ABB RAPID module: PathProbe.mod

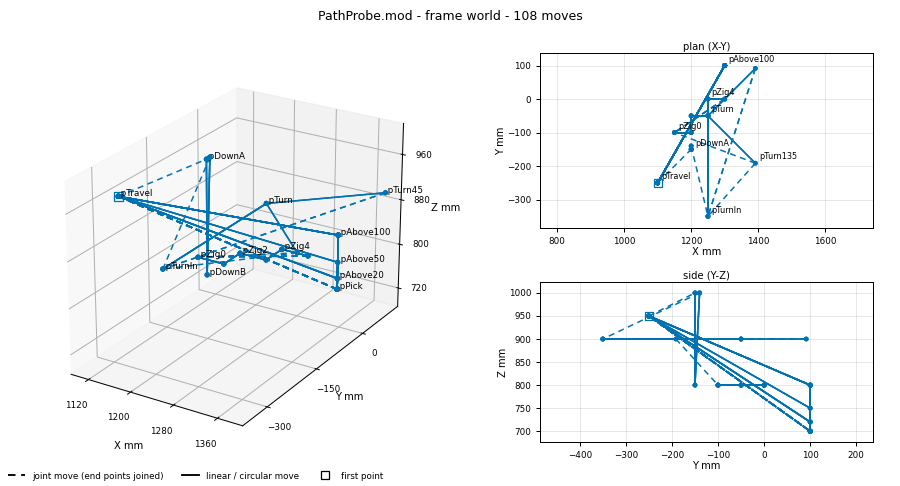
[picture p0: tool path of PathProbe.mod in frame world, 108 of 108 moves have a stored position in this frame; points joined in program order, loops and branches not executed]
MODULE PathProbe
    ! CrossArm - path probe. PROC Path runs every move CrossArm converts; the TCP is read while it moves.
    CONST robtarget pTravel:=[[1100,-250,950],[0,0.3826834,0.9238795,0],[-1,0,0,0],[9E+09,9E+09,9E+09,9E+09,9E+09,9E+09]];
    CONST robtarget pPick:=[[1300,100,700],[0,0.3826834,0.9238795,0],[0,0,0,0],[9E+09,9E+09,9E+09,9E+09,9E+09,9E+09]];
    CONST robtarget pAbove100:=[[1300,100,800],[0,0.3826834,0.9238795,0],[0,0,0,0],[9E+09,9E+09,9E+09,9E+09,9E+09,9E+09]];
    CONST robtarget pAbove50:=[[1300,100,750],[0,0.3826834,0.9238795,0],[0,0,0,0],[9E+09,9E+09,9E+09,9E+09,9E+09,9E+09]];
    CONST robtarget pAbove20:=[[1300,100,720],[0,0.3826834,0.9238795,0],[0,0,0,0],[9E+09,9E+09,9E+09,9E+09,9E+09,9E+09]];
    CONST robtarget pDownA:=[[1200,-150,1000],[0,0.3826834,0.9238795,0],[-1,0,0,0],[9E+09,9E+09,9E+09,9E+09,9E+09,9E+09]];
    CONST robtarget pDownB:=[[1200,-150,800],[0,0.3826834,0.9238795,0],[-1,0,0,0],[9E+09,9E+09,9E+09,9E+09,9E+09,9E+09]];
    CONST robtarget pDownC:=[[1200,-140,1000],[0,0.3826834,0.9238795,0],[-1,0,0,0],[9E+09,9E+09,9E+09,9E+09,9E+09,9E+09]];
    CONST robtarget pTurnIn:=[[1250,-350,900],[0,0.3826834,0.9238795,0],[-1,0,0,0],[9E+09,9E+09,9E+09,9E+09,9E+09,9E+09]];
    CONST robtarget pTurn:=[[1250,-50,900],[0,0.3826834,0.9238795,0],[-1,0,0,0],[9E+09,9E+09,9E+09,9E+09,9E+09,9E+09]];
    CONST robtarget pTurn45:=[[1391.421,91.421,900],[0,0.3826834,0.9238795,0],[0,0,0,0],[9E+09,9E+09,9E+09,9E+09,9E+09,9E+09]];
    CONST robtarget pTurn135:=[[1391.421,-191.421,900],[0,0.3826834,0.9238795,0],[-1,0,0,0],[9E+09,9E+09,9E+09,9E+09,9E+09,9E+09]];
    CONST robtarget pZig0:=[[1150,-100,800],[0,0.3826834,0.9238795,0],[-1,0,0,0],[9E+09,9E+09,9E+09,9E+09,9E+09,9E+09]];
    CONST robtarget pZig1:=[[1200,-100,800],[0,0.3826834,0.9238795,0],[-1,0,0,0],[9E+09,9E+09,9E+09,9E+09,9E+09,9E+09]];
    CONST robtarget pZig2:=[[1200,-50,800],[0,0.3826834,0.9238795,0],[-1,0,0,0],[9E+09,9E+09,9E+09,9E+09,9E+09,9E+09]];
    CONST robtarget pZig3:=[[1250,-50,800],[0,0.3826834,0.9238795,0],[-1,0,0,0],[9E+09,9E+09,9E+09,9E+09,9E+09,9E+09]];
    CONST robtarget pZig4:=[[1250,0,800],[0,0.3826834,0.9238795,0],[0,0,0,0],[9E+09,9E+09,9E+09,9E+09,9E+09,9E+09]];
    CONST robtarget pZig5:=[[1300,0,800],[0,0.3826834,0.9238795,0],[0,0,0,0],[9E+09,9E+09,9E+09,9E+09,9E+09,9E+09]];

    PROC Path()
        MoveJ pTravel,v1000,fine,tool0;
        MoveL pAbove100,v1000,z10,tool0;
        MoveL pPick,v300,fine,tool0;
        MoveJ pTravel,v1000,fine,tool0;
        MoveL pAbove100,v1000,z50,tool0;
        MoveL pPick,v300,fine,tool0;
        MoveJ pTravel,v1000,fine,tool0;
        MoveL pAbove100,v1000,z100,tool0;
        MoveL pPick,v300,fine,tool0;
        MoveJ pTravel,v1000,fine,tool0;
        MoveL pAbove50,v1000,z10,tool0;
        MoveL pPick,v300,fine,tool0;
        MoveJ pTravel,v1000,fine,tool0;
        MoveL pAbove50,v1000,z50,tool0;
        MoveL pPick,v300,fine,tool0;
        MoveJ pTravel,v1000,fine,tool0;
        MoveL pAbove50,v1000,z100,tool0;
        MoveL pPick,v300,fine,tool0;
        MoveJ pTravel,v1000,fine,tool0;
        MoveL pAbove20,v1000,z10,tool0;
        MoveL pPick,v300,fine,tool0;
        MoveJ pTravel,v1000,fine,tool0;
        MoveL pAbove20,v1000,z50,tool0;
        MoveL pPick,v300,fine,tool0;
        MoveJ pTravel,v1000,fine,tool0;
        MoveL pAbove20,v1000,z100,tool0;
        MoveL pPick,v300,fine,tool0;
        MoveJ pTravel,v1000,fine,tool0;
        MoveJ pAbove100,v1000,z10,tool0;
        MoveL pPick,v300,fine,tool0;
        MoveJ pTravel,v1000,fine,tool0;
        MoveJ pAbove100,v1000,z50,tool0;
        MoveL pPick,v300,fine,tool0;
        MoveJ pTravel,v1000,fine,tool0;
        MoveJ pAbove100,v1000,z100,tool0;
        MoveL pPick,v300,fine,tool0;
        MoveJ pPick,v1000,fine,tool0;
        MoveL pAbove100,v300,z10,tool0;
        MoveL pTravel,v1000,fine,tool0;
        MoveJ pPick,v1000,fine,tool0;
        MoveL pAbove100,v300,z50,tool0;
        MoveL pTravel,v1000,fine,tool0;
        MoveJ pPick,v1000,fine,tool0;
        MoveL pAbove100,v300,z100,tool0;
        MoveL pTravel,v1000,fine,tool0;
        MoveJ pPick,v1000,fine,tool0;
        MoveL pAbove20,v300,z10,tool0;
        MoveL pTravel,v1000,fine,tool0;
        MoveJ pPick,v1000,fine,tool0;
        MoveL pAbove20,v300,z50,tool0;
        MoveL pTravel,v1000,fine,tool0;
        MoveJ pPick,v1000,fine,tool0;
        MoveL pAbove20,v300,z100,tool0;
        MoveL pTravel,v1000,fine,tool0;
        MoveJ pPick,v1000,fine,tool0;
        MoveL pAbove100,v300,z10,tool0;
        MoveJ pTravel,v1000,fine,tool0;
        MoveJ pPick,v1000,fine,tool0;
        MoveL pAbove100,v300,z50,tool0;
        MoveJ pTravel,v1000,fine,tool0;
        MoveJ pPick,v1000,fine,tool0;
        MoveL pAbove100,v300,z100,tool0;
        MoveJ pTravel,v1000,fine,tool0;
        MoveJ pDownA,v1000,fine,tool0;
        MoveL pDownB,v600,z5,tool0;
        MoveL pDownC,v600,fine,tool0;
        MoveJ pDownA,v1000,fine,tool0;
        MoveL pDownB,v600,z20,tool0;
        MoveL pDownC,v600,fine,tool0;
        MoveJ pDownA,v1000,fine,tool0;
        MoveL pDownB,v600,z50,tool0;
        MoveL pDownC,v600,fine,tool0;
        MoveJ pTurnIn,v1000,fine,tool0;
        MoveL pTurn,v600,z10,tool0;
        MoveL pTurn45,v600,fine,tool0;
        MoveJ pTurnIn,v1000,fine,tool0;
        MoveL pTurn,v600,z50,tool0;
        MoveL pTurn45,v600,fine,tool0;
        MoveJ pTurnIn,v1000,fine,tool0;
        MoveL pTurn,v600,z10,tool0;
        MoveL pTurn135,v600,fine,tool0;
        MoveJ pTurnIn,v1000,fine,tool0;
        MoveL pTurn,v600,z50,tool0;
        MoveL pTurn135,v600,fine,tool0;
        MoveJ pZig0,v1000,fine,tool0;
        MoveL pZig1,v300,z10,tool0;
        MoveL pZig2,v300,z10,tool0;
        MoveL pZig3,v300,z10,tool0;
        MoveL pZig4,v300,z10,tool0;
        MoveL pZig5,v300,fine,tool0;
        MoveJ pZig0,v1000,fine,tool0;
        MoveL pZig1,v300,z20,tool0;
        MoveL pZig2,v300,z20,tool0;
        MoveL pZig3,v300,z20,tool0;
        MoveL pZig4,v300,z20,tool0;
        MoveL pZig5,v300,fine,tool0;
        MoveJ pZig0,v1000,fine,tool0;
        MoveL pZig1,v600,z10,tool0;
        MoveL pZig2,v600,z10,tool0;
        MoveL pZig3,v600,z10,tool0;
        MoveL pZig4,v600,z10,tool0;
        MoveL pZig5,v600,fine,tool0;
        MoveJ pZig0,v1000,fine,tool0;
        MoveL pZig1,v600,z20,tool0;
        MoveL pZig2,v600,z20,tool0;
        MoveL pZig3,v600,z20,tool0;
        MoveL pZig4,v600,z20,tool0;
        MoveL pZig5,v600,fine,tool0;
    ENDPROC
ENDMODULE
